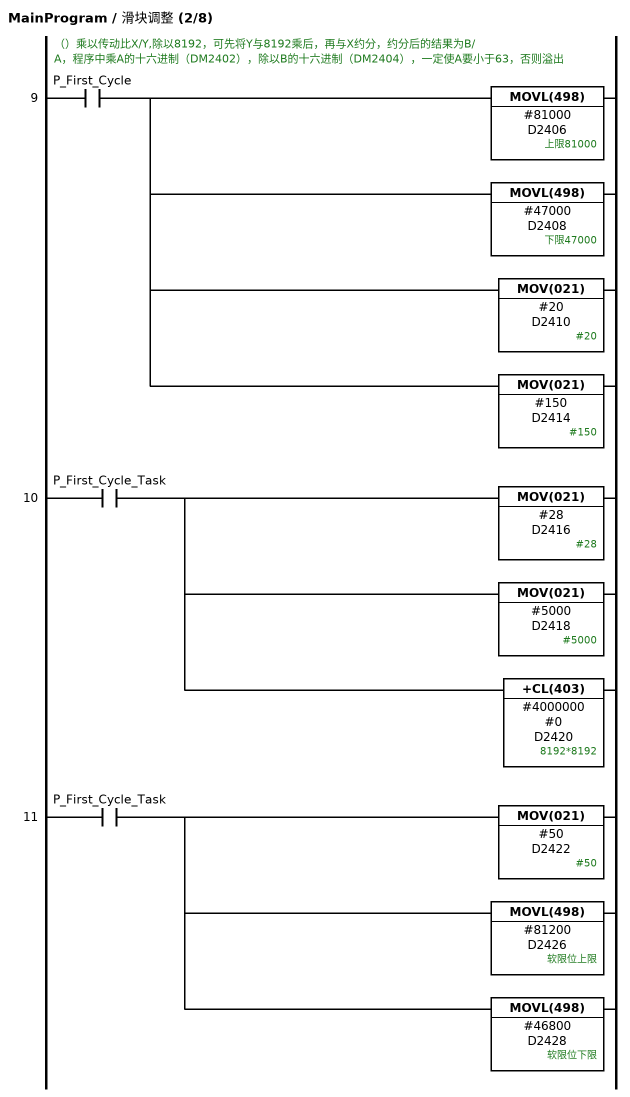
; [picture p24: MainProgram / 滑块调整, rungs 9-11]
; rung 9: （）乘以传动比X/Y,除以8192，可先将Y与8192乘后，再与X约分，约分后的结果为B/A，程序中乘A的十六进制（DM2402），除以B的十六进制（DM2404），一定使A要小于63，否则溢出
LD P_First_Cycle
MOVL(498) #81000 D2406  ; 上限81000
MOVL(498) #47000 D2408  ; 下限47000
MOV(021) #20 D2410  ; #20
MOV(021) #150 D2414  ; #150
; rung 10
LD P_First_Cycle_Task
MOV(021) #28 D2416  ; #28
MOV(021) #5000 D2418  ; #5000
+CL(403) #4000000 #0 D2420  ; 8192*8192
; rung 11
LD P_First_Cycle_Task
MOV(021) #50 D2422  ; #50
MOVL(498) #81200 D2426  ; 软限位上限
MOVL(498) #46800 D2428  ; 软限位下限

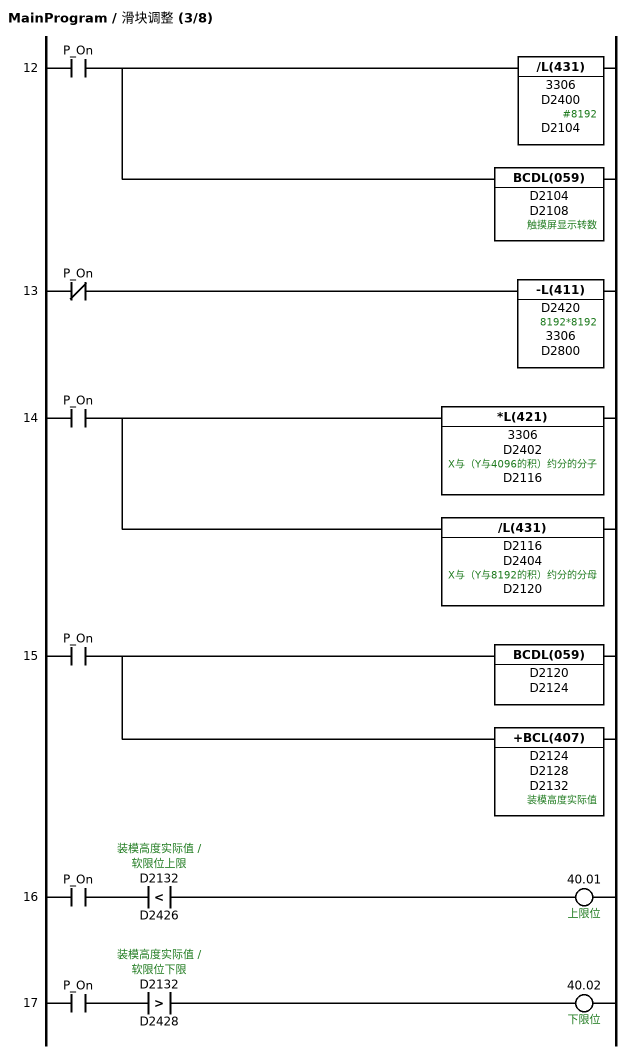
; rung 12
LD P_On
/L(431) 3306 D2400 D2104  ; #8192
BCDL(059) D2104 D2108  ; 触摸屏显示转数
; rung 13
LDNOT P_On
-L(411) D2420 3306 D2800  ; 8192*8192
; rung 14
LD P_On
*L(421) 3306 D2402 D2116  ; X与（Y与4096的积）约分的分子
/L(431) D2116 D2404 D2120  ; X与（Y与8192的积）约分的分母
; rung 15
LD P_On
BCDL(059) D2120 D2124
+BCL(407) D2124 D2128 D2132  ; 装模高度实际值
; rung 16
LD P_On
AND<L(311) D2132 D2426  ; 装模高度实际值, 软限位上限
OUT 40.01  ; 上限位
; rung 17
LD P_On
AND>L(321) D2132 D2428  ; 装模高度实际值, 软限位下限
OUT 40.02  ; 下限位

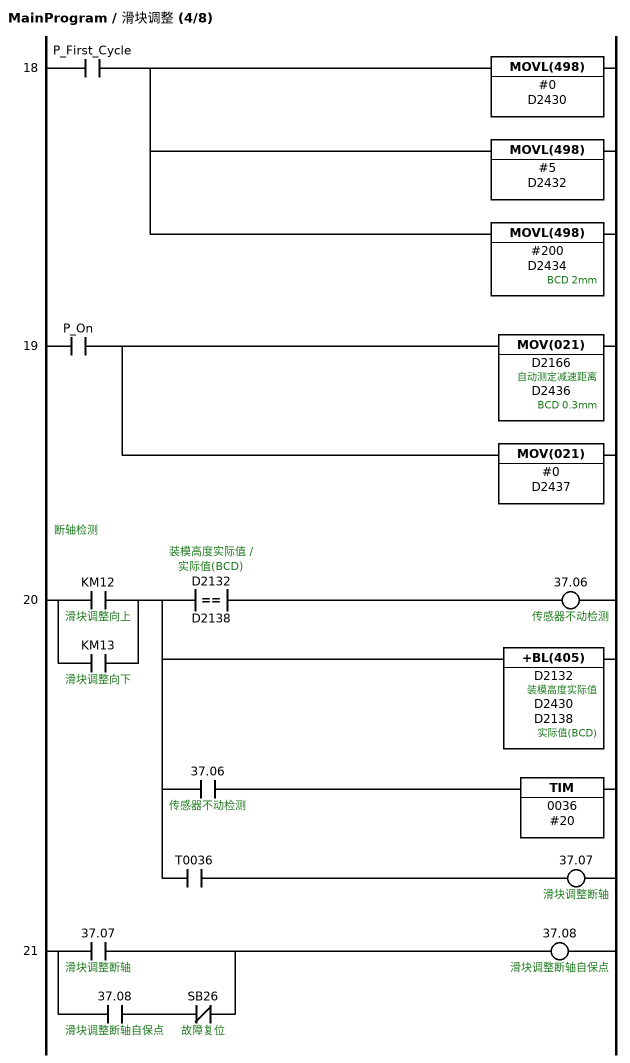
; rung 18
LD P_First_Cycle
MOVL(498) #0 D2430
MOVL(498) #5 D2432
MOVL(498) #200 D2434  ; BCD 2mm
; rung 19
LD P_On
MOV(021) D2166 D2436  ; 自动测定减速距离, BCD 0.3mm
MOV(021) #0 D2437
; rung 20: 断轴检测
LD KM12  ; 滑块调整向上
OR KM13  ; 滑块调整向下
OUT TR0
AND=L(301) D2132 D2138  ; 装模高度实际值, 实际值(BCD)
OUT 37.06  ; 传感器不动检测
LD TR0
+BL(405) D2132 D2430 D2138  ; 装模高度实际值, 实际值(BCD)
AND 37.06  ; 传感器不动检测
TIM 0036 #20
LD TR0
AND T0036
OUT 37.07  ; 滑块调整断轴
; rung 21
LD 37.07  ; 滑块调整断轴
LD 37.08  ; 滑块调整断轴自保点
ANDNOT SB26  ; 故障复位
ORLD
OUT 37.08  ; 滑块调整断轴自保点

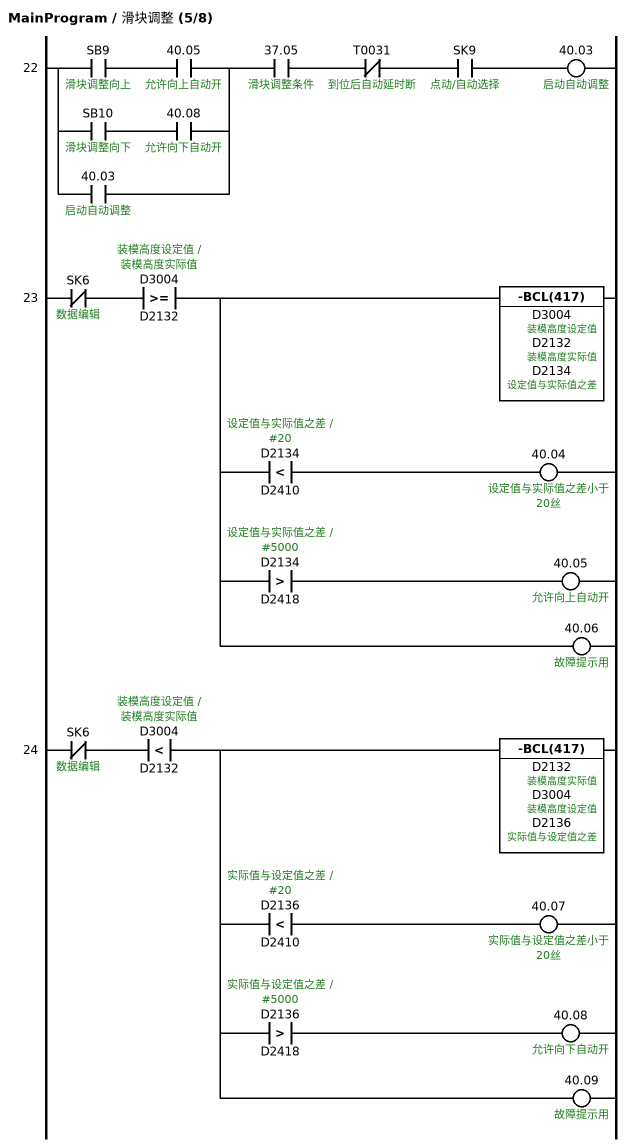
; rung 22
LD SB9  ; 滑块调整向上
AND 40.05  ; 允许向上自动开
LD SB10  ; 滑块调整向下
AND 40.08  ; 允许向下自动开
ORLD
OR 40.03  ; 启动自动调整
AND 37.05  ; 滑块调整条件
ANDNOT T0031  ; 到位后自动延时断
AND SK9  ; 点动/自动选择
OUT 40.03  ; 启动自动调整
; rung 23
LDNOT SK6  ; 数据编辑
AND>=L(326) D3004 D2132  ; 装模高度设定值, 装模高度实际值
OUT TR0
-BCL(417) D3004 D2132 D2134  ; 装模高度设定值, 装模高度实际值, 设定值与实际值之差
AND<L(311) D2134 D2410  ; 设定值与实际值之差, #20
OUT 40.04  ; 设定值与实际值之差小于20丝
LD TR0
AND>L(321) D2134 D2418  ; 设定值与实际值之差, #5000
OUT 40.05  ; 允许向上自动开
LD TR0
OUT 40.06  ; 故障提示用
; rung 24
LDNOT SK6  ; 数据编辑
AND<L(311) D3004 D2132  ; 装模高度设定值, 装模高度实际值
OUT TR0
-BCL(417) D2132 D3004 D2136  ; 装模高度实际值, 装模高度设定值, 实际值与设定值之差
AND<L(311) D2136 D2410  ; 实际值与设定值之差, #20
OUT 40.07  ; 实际值与设定值之差小于20丝
LD TR0
AND>L(321) D2136 D2418  ; 实际值与设定值之差, #5000
OUT 40.08  ; 允许向下自动开
LD TR0
OUT 40.09  ; 故障提示用

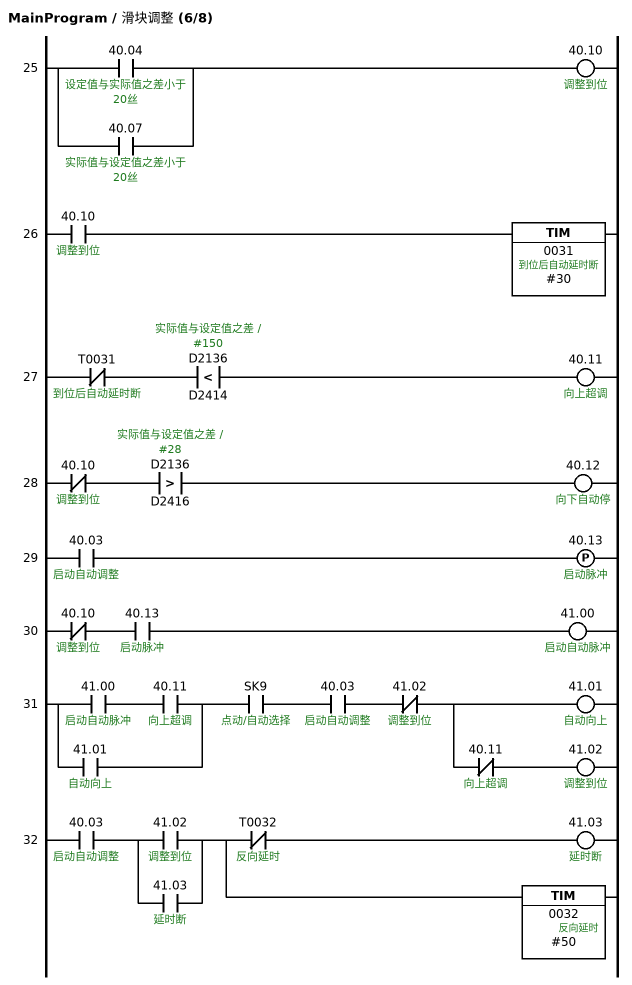
; rung 25
LD 40.04  ; 设定值与实际值之差小于20丝
OR 40.07  ; 实际值与设定值之差小于20丝
OUT 40.10  ; 调整到位
; rung 26
LD 40.10  ; 调整到位
TIM 0031 #30  ; 到位后自动延时断
; rung 27
LDNOT T0031  ; 到位后自动延时断
AND<L(311) D2136 D2414  ; 实际值与设定值之差, #150
OUT 40.11  ; 向上超调
; rung 28
LDNOT 40.10  ; 调整到位
AND>L(321) D2136 D2416  ; 实际值与设定值之差, #28
OUT 40.12  ; 向下自动停
; rung 29
LD 40.03  ; 启动自动调整
DIFU(013) 40.13  ; 启动脉冲
; rung 30
LDNOT 40.10  ; 调整到位
AND 40.13  ; 启动脉冲
OUT 41.00  ; 启动自动脉冲
; rung 31
LD 41.00  ; 启动自动脉冲
AND 40.11  ; 向上超调
OR 41.01  ; 自动向上
AND SK9  ; 点动/自动选择
AND 40.03  ; 启动自动调整
ANDNOT 41.02  ; 调整到位
OUT 41.01  ; 自动向上
ANDNOT 40.11  ; 向上超调
OUT 41.02  ; 调整到位
; rung 32
LD 40.03  ; 启动自动调整
LD 41.02  ; 调整到位
OR 41.03  ; 延时断
ANDLD
OUT TR0
ANDNOT T0032  ; 反向延时
OUT 41.03  ; 延时断
LD TR0
TIM 0032 #50  ; 反向延时

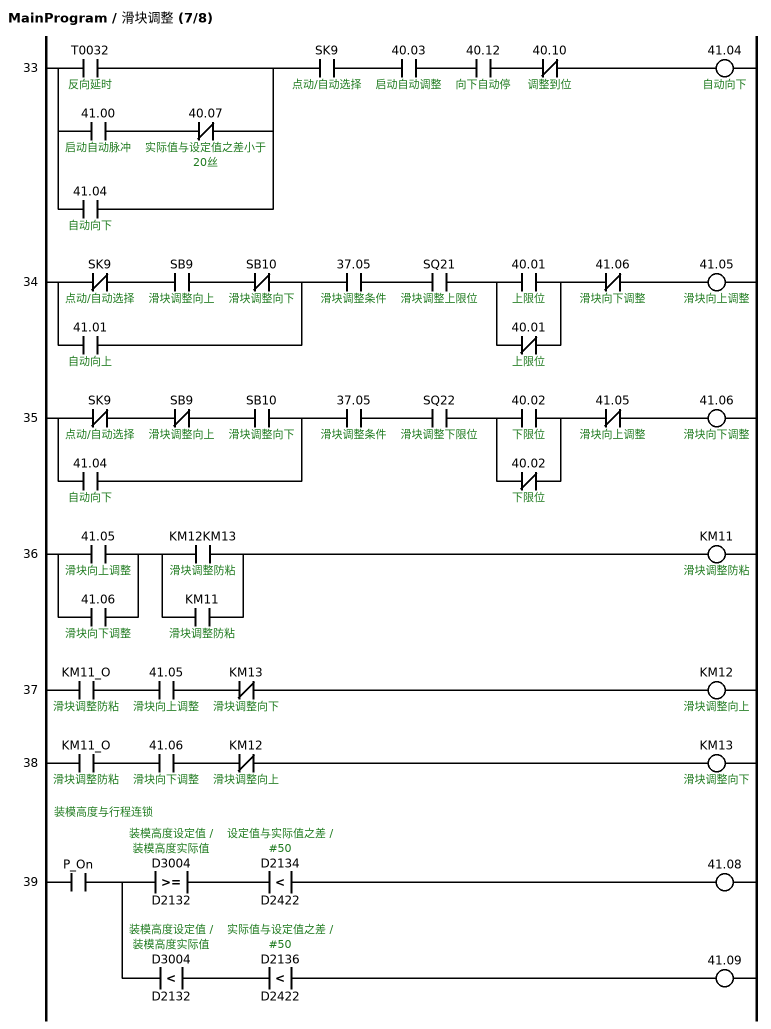
; rung 33
LD T0032  ; 反向延时
LD 41.00  ; 启动自动脉冲
ANDNOT 40.07  ; 实际值与设定值之差小于20丝
ORLD
OR 41.04  ; 自动向下
AND SK9  ; 点动/自动选择
AND 40.03  ; 启动自动调整
AND 40.12  ; 向下自动停
ANDNOT 40.10  ; 调整到位
OUT 41.04  ; 自动向下
; rung 34
LDNOT SK9  ; 点动/自动选择
AND SB9  ; 滑块调整向上
ANDNOT SB10  ; 滑块调整向下
OR 41.01  ; 自动向上
AND 37.05  ; 滑块调整条件
AND SQ21  ; 滑块调整上限位
LD 40.01  ; 上限位
ORNOT 40.01  ; 上限位
ANDLD
ANDNOT 41.06  ; 滑块向下调整
OUT 41.05  ; 滑块向上调整
; rung 35
LDNOT SK9  ; 点动/自动选择
ANDNOT SB9  ; 滑块调整向上
AND SB10  ; 滑块调整向下
OR 41.04  ; 自动向下
AND 37.05  ; 滑块调整条件
AND SQ22  ; 滑块调整下限位
LD 40.02  ; 下限位
ORNOT 40.02  ; 下限位
ANDLD
ANDNOT 41.05  ; 滑块向上调整
OUT 41.06  ; 滑块向下调整
; rung 36
LD 41.05  ; 滑块向上调整
OR 41.06  ; 滑块向下调整
LD KM12KM13  ; 滑块调整防粘
OR KM11  ; 滑块调整防粘
ANDLD
OUT KM11  ; 滑块调整防粘
; rung 37
LD KM11_O  ; 滑块调整防粘
AND 41.05  ; 滑块向上调整
ANDNOT KM13  ; 滑块调整向下
OUT KM12  ; 滑块调整向上
; rung 38
LD KM11_O  ; 滑块调整防粘
AND 41.06  ; 滑块向下调整
ANDNOT KM12  ; 滑块调整向上
OUT KM13  ; 滑块调整向下
; rung 39: 装模高度与行程连锁
LD P_On
OUT TR0
AND>=L(326) D3004 D2132  ; 装模高度设定值, 装模高度实际值
AND<L(311) D2134 D2422  ; 设定值与实际值之差, #50
OUT 41.08
LD TR0
AND<L(311) D3004 D2132  ; 装模高度设定值, 装模高度实际值
AND<L(311) D2136 D2422  ; 实际值与设定值之差, #50
OUT 41.09

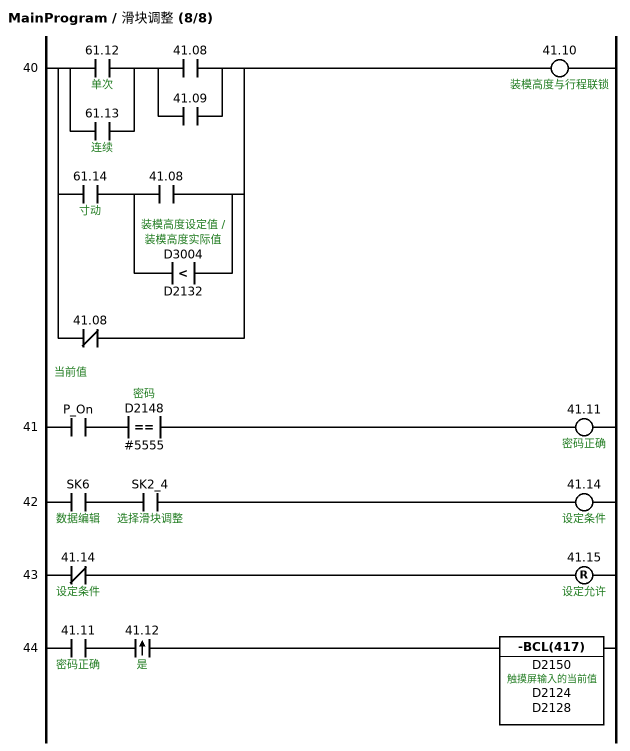
; rung 40
LD 61.12  ; 单次
OR 61.13  ; 连续
LD 41.08
OR 41.09
ANDLD
LD 61.14  ; 寸动
LD 41.08
OR<L(311) D3004 D2132  ; 装模高度设定值, 装模高度实际值
ANDLD
ORLD
ORNOT 41.08
OUT 41.10  ; 装模高度与行程联锁
; rung 41: 当前值
LD P_On
AND=(300) D2148 #5555  ; 密码
OUT 41.11  ; 密码正确
; rung 42
LD SK6  ; 数据编辑
AND SK2_4  ; 选择滑块调整
OUT 41.14  ; 设定条件
; rung 43
LDNOT 41.14  ; 设定条件
RSET 41.15  ; 设定允许
; rung 44
LD 41.11  ; 密码正确
@AND 41.12  ; 是
-BCL(417) D2150 D2124 D2128  ; 触摸屏输入的当前值

### Section 气垫调整

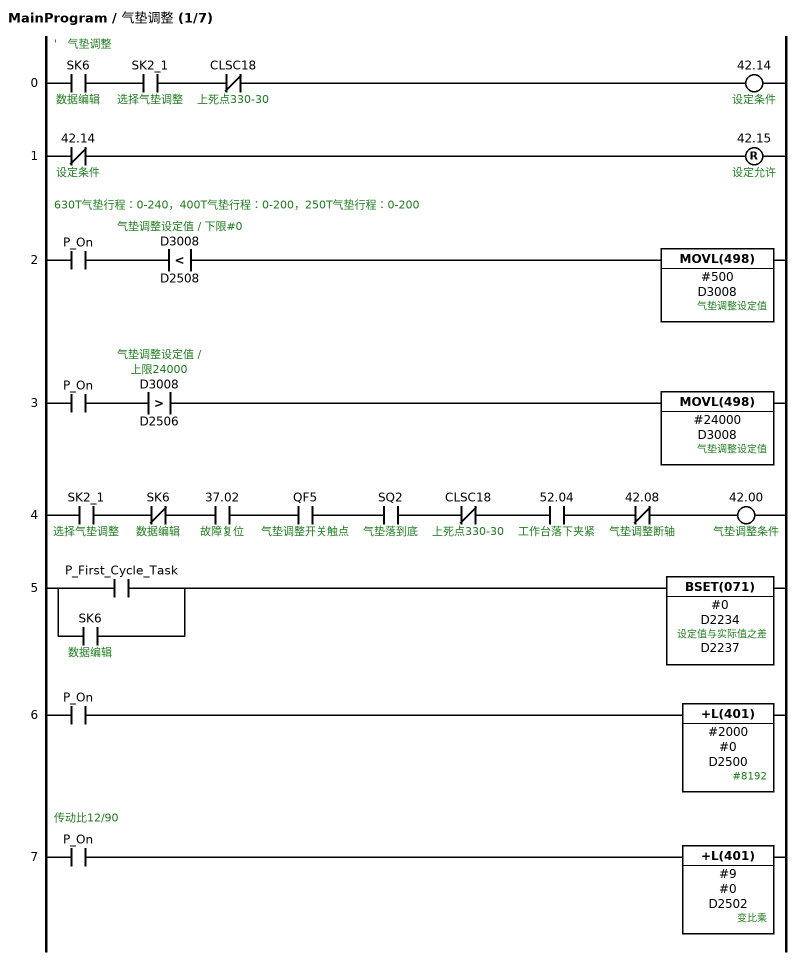
; rung 0: '   气垫调整
LD SK6  ; 数据编辑
AND SK2_1  ; 选择气垫调整
ANDNOT CLSC18  ; 上死点330-30
OUT 42.14  ; 设定条件
; rung 1
LDNOT 42.14  ; 设定条件
RSET 42.15  ; 设定允许
; rung 2: 630T气垫行程：0-240，400T气垫行程：0-200，250T气垫行程：0-200
LD P_On
AND<L(311) D3008 D2508  ; 气垫调整设定值, 下限#0
MOVL(498) #500 D3008  ; 气垫调整设定值
; rung 3
LD P_On
AND>L(321) D3008 D2506  ; 气垫调整设定值, 上限24000
MOVL(498) #24000 D3008  ; 气垫调整设定值
; rung 4
LD SK2_1  ; 选择气垫调整
ANDNOT SK6  ; 数据编辑
AND 37.02  ; 故障复位
AND QF5  ; 气垫调整开关触点
AND SQ2  ; 气垫落到底
ANDNOT CLSC18  ; 上死点330-30
AND 52.04  ; 工作台落下夹紧
ANDNOT 42.08  ; 气垫调整断轴
OUT 42.00  ; 气垫调整条件
; rung 5
LD P_First_Cycle_Task
OR SK6  ; 数据编辑
BSET(071) #0 D2234 D2237  ; 设定值与实际值之差
; rung 6
LD P_On
+L(401) #2000 #0 D2500  ; #8192
; rung 7: 传动比12/90
LD P_On
+L(401) #9 #0 D2502  ; 变比乘

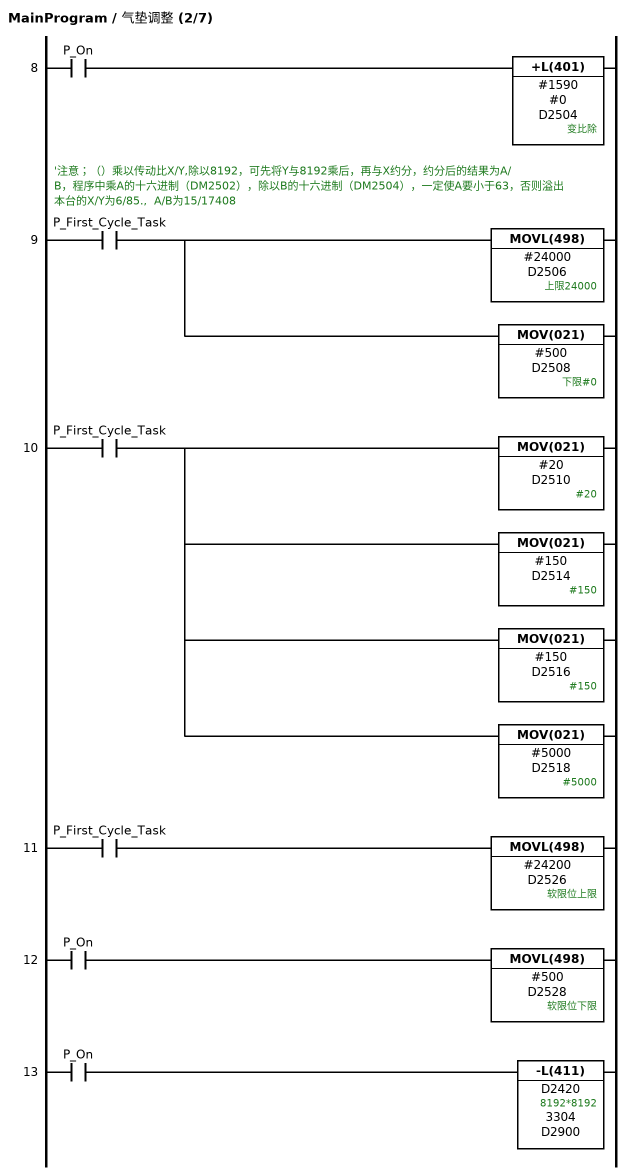
; rung 8
LD P_On
+L(401) #1590 #0 D2504  ; 变比除
; rung 9: '注意；（）乘以传动比X/Y,除以8192，可先将Y与8192乘后，再与X约分，约分后的结果为A/B，程序中乘A的十六进制（DM2502），除以B的十六进制（DM2504），一定使A要小于63，否则溢出                本台的X/Y为6/85.,  A/B为15/17408
LD P_First_Cycle_Task
MOVL(498) #24000 D2506  ; 上限24000
MOV(021) #500 D2508  ; 下限#0
; rung 10
LD P_First_Cycle_Task
MOV(021) #20 D2510  ; #20
MOV(021) #150 D2514  ; #150
MOV(021) #150 D2516  ; #150
MOV(021) #5000 D2518  ; #5000
; rung 11
LD P_First_Cycle_Task
MOVL(498) #24200 D2526  ; 软限位上限
; rung 12
LD P_On
MOVL(498) #500 D2528  ; 软限位下限
; rung 13
LD P_On
-L(411) D2420 3304 D2900  ; 8192*8192

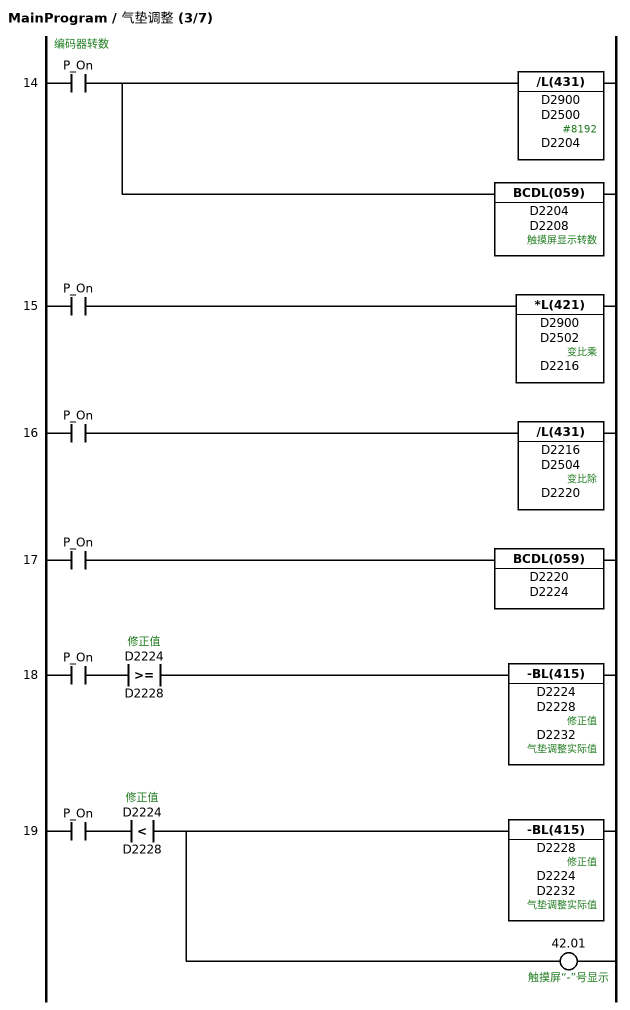
; rung 14: 编码器转数
LD P_On
/L(431) D2900 D2500 D2204  ; #8192
BCDL(059) D2204 D2208  ; 触摸屏显示转数
; rung 15
LD P_On
*L(421) D2900 D2502 D2216  ; 变比乘
; rung 16
LD P_On
/L(431) D2216 D2504 D2220  ; 变比除
; rung 17
LD P_On
BCDL(059) D2220 D2224
; rung 18
LD P_On
AND>=L(326) D2224 D2228  ; 修正值
-BL(415) D2224 D2228 D2232  ; 修正值, 气垫调整实际值
; rung 19
LD P_On
AND<L(311) D2224 D2228  ; 修正值
-BL(415) D2228 D2224 D2232  ; 修正值, 气垫调整实际值
OUT 42.01  ; 触摸屏“-”号显示

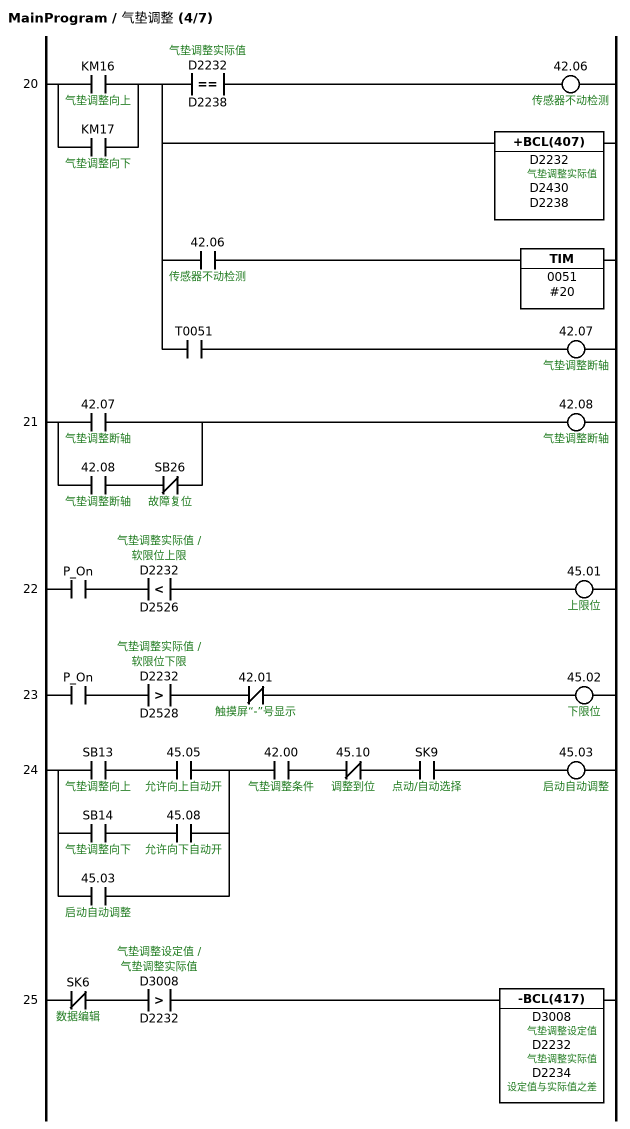
; rung 20
LD KM16  ; 气垫调整向上
OR KM17  ; 气垫调整向下
OUT TR0
AND=L(301) D2232 D2238  ; 气垫调整实际值
OUT 42.06  ; 传感器不动检测
LD TR0
+BCL(407) D2232 D2430 D2238  ; 气垫调整实际值
AND 42.06  ; 传感器不动检测
TIM 0051 #20
LD TR0
AND T0051
OUT 42.07  ; 气垫调整断轴
; rung 21
LD 42.07  ; 气垫调整断轴
LD 42.08  ; 气垫调整断轴
ANDNOT SB26  ; 故障复位
ORLD
OUT 42.08  ; 气垫调整断轴
; rung 22
LD P_On
AND<L(311) D2232 D2526  ; 气垫调整实际值, 软限位上限
OUT 45.01  ; 上限位
; rung 23
LD P_On
AND>L(321) D2232 D2528  ; 气垫调整实际值, 软限位下限
ANDNOT 42.01  ; 触摸屏“-”号显示
OUT 45.02  ; 下限位
; rung 24
LD SB13  ; 气垫调整向上
AND 45.05  ; 允许向上自动开
LD SB14  ; 气垫调整向下
AND 45.08  ; 允许向下自动开
ORLD
OR 45.03  ; 启动自动调整
AND 42.00  ; 气垫调整条件
ANDNOT 45.10  ; 调整到位
AND SK9  ; 点动/自动选择
OUT 45.03  ; 启动自动调整
; rung 25
LDNOT SK6  ; 数据编辑
AND>L(321) D3008 D2232  ; 气垫调整设定值, 气垫调整实际值
-BCL(417) D3008 D2232 D2234  ; 气垫调整设定值, 气垫调整实际值, 设定值与实际值之差

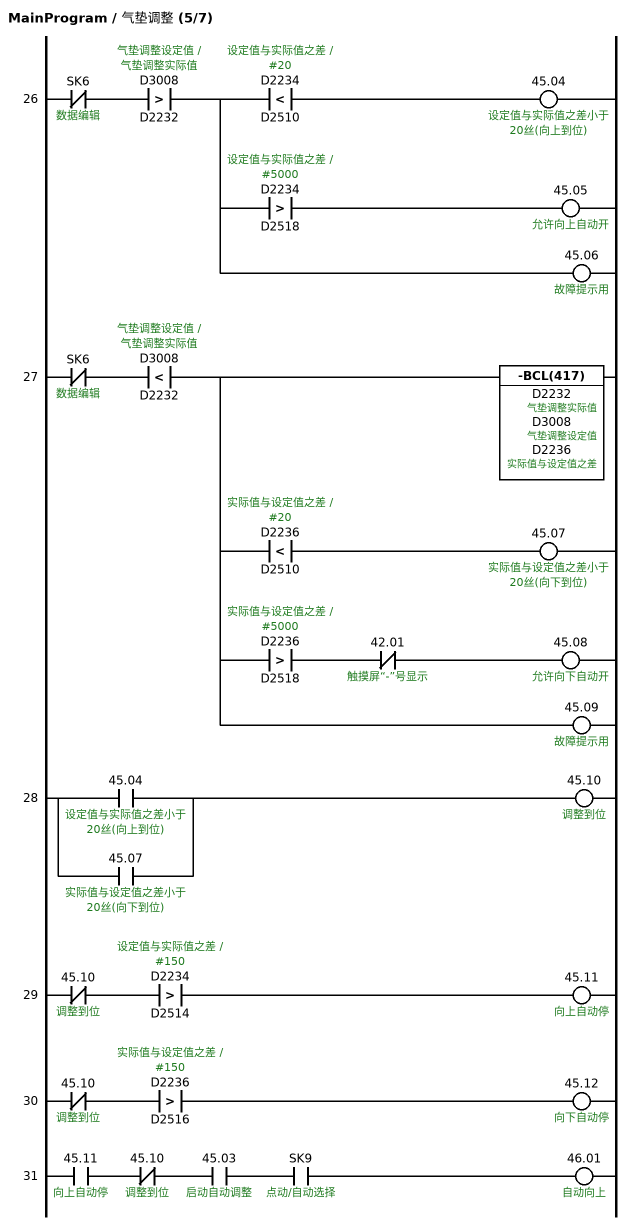
; rung 26
LDNOT SK6  ; 数据编辑
AND>L(321) D3008 D2232  ; 气垫调整设定值, 气垫调整实际值
OUT TR0
AND<L(311) D2234 D2510  ; 设定值与实际值之差, #20
OUT 45.04  ; 设定值与实际值之差小于20丝(向上到位)
LD TR0
AND>L(321) D2234 D2518  ; 设定值与实际值之差, #5000
OUT 45.05  ; 允许向上自动开
LD TR0
OUT 45.06  ; 故障提示用
; rung 27
LDNOT SK6  ; 数据编辑
AND<L(311) D3008 D2232  ; 气垫调整设定值, 气垫调整实际值
OUT TR0
-BCL(417) D2232 D3008 D2236  ; 气垫调整实际值, 气垫调整设定值, 实际值与设定值之差
AND<L(311) D2236 D2510  ; 实际值与设定值之差, #20
OUT 45.07  ; 实际值与设定值之差小于20丝(向下到位)
LD TR0
AND>L(321) D2236 D2518  ; 实际值与设定值之差, #5000
ANDNOT 42.01  ; 触摸屏“-”号显示
OUT 45.08  ; 允许向下自动开
LD TR0
OUT 45.09  ; 故障提示用
; rung 28
LD 45.04  ; 设定值与实际值之差小于20丝(向上到位)
OR 45.07  ; 实际值与设定值之差小于20丝(向下到位)
OUT 45.10  ; 调整到位
; rung 29
LDNOT 45.10  ; 调整到位
AND>L(321) D2234 D2514  ; 设定值与实际值之差, #150
OUT 45.11  ; 向上自动停
; rung 30
LDNOT 45.10  ; 调整到位
AND>L(321) D2236 D2516  ; 实际值与设定值之差, #150
OUT 45.12  ; 向下自动停
; rung 31
LD 45.11  ; 向上自动停
ANDNOT 45.10  ; 调整到位
AND 45.03  ; 启动自动调整
AND SK9  ; 点动/自动选择
OUT 46.01  ; 自动向上

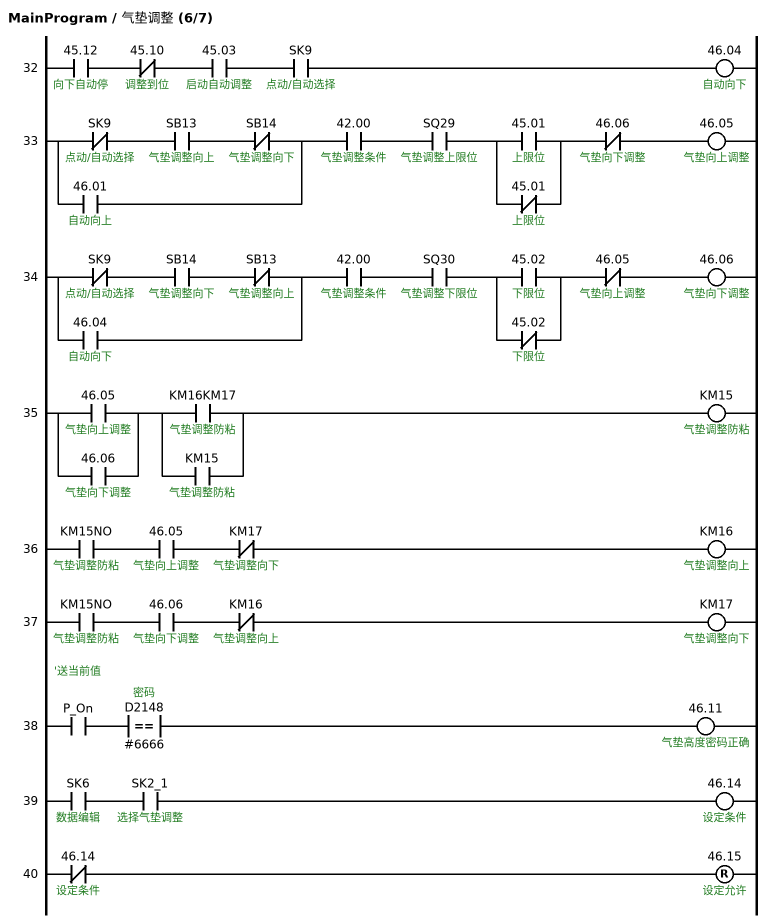
; rung 32
LD 45.12  ; 向下自动停
ANDNOT 45.10  ; 调整到位
AND 45.03  ; 启动自动调整
AND SK9  ; 点动/自动选择
OUT 46.04  ; 自动向下
; rung 33
LDNOT SK9  ; 点动/自动选择
AND SB13  ; 气垫调整向上
ANDNOT SB14  ; 气垫调整向下
OR 46.01  ; 自动向上
AND 42.00  ; 气垫调整条件
AND SQ29  ; 气垫调整上限位
LD 45.01  ; 上限位
ORNOT 45.01  ; 上限位
ANDLD
ANDNOT 46.06  ; 气垫向下调整
OUT 46.05  ; 气垫向上调整
; rung 34
LDNOT SK9  ; 点动/自动选择
AND SB14  ; 气垫调整向下
ANDNOT SB13  ; 气垫调整向上
OR 46.04  ; 自动向下
AND 42.00  ; 气垫调整条件
AND SQ30  ; 气垫调整下限位
LD 45.02  ; 下限位
ORNOT 45.02  ; 下限位
ANDLD
ANDNOT 46.05  ; 气垫向上调整
OUT 46.06  ; 气垫向下调整
; rung 35
LD 46.05  ; 气垫向上调整
OR 46.06  ; 气垫向下调整
LD KM16KM17  ; 气垫调整防粘
OR KM15  ; 气垫调整防粘
ANDLD
OUT KM15  ; 气垫调整防粘
; rung 36
LD KM15NO  ; 气垫调整防粘
AND 46.05  ; 气垫向上调整
ANDNOT KM17  ; 气垫调整向下
OUT KM16  ; 气垫调整向上
; rung 37
LD KM15NO  ; 气垫调整防粘
AND 46.06  ; 气垫向下调整
ANDNOT KM16  ; 气垫调整向上
OUT KM17  ; 气垫调整向下
; rung 38: '送当前值
LD P_On
AND=L(301) D2148 #6666  ; 密码
OUT 46.11  ; 气垫高度密码正确
; rung 39
LD SK6  ; 数据编辑
AND SK2_1  ; 选择气垫调整
OUT 46.14  ; 设定条件
; rung 40
LDNOT 46.14  ; 设定条件
RSET 46.15  ; 设定允许

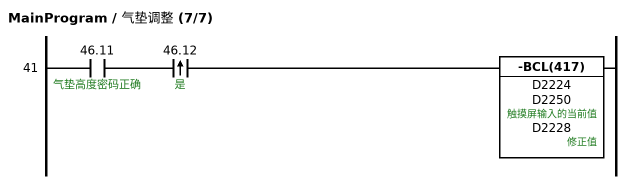
; rung 41
LD 46.11  ; 气垫高度密码正确
@AND 46.12  ; 是
-BCL(417) D2224 D2250 D2228  ; 触摸屏输入的当前值, 修正值

### Section 气垫顶起

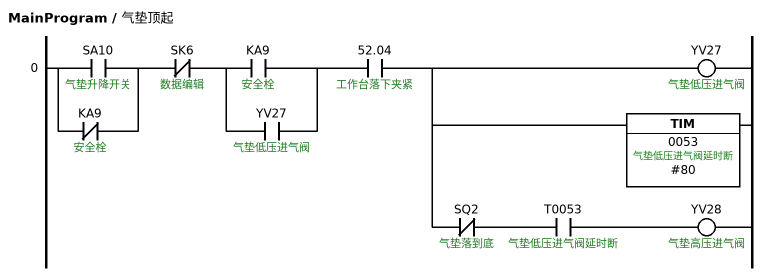
; rung 0
LD SA10  ; 气垫升降开关
ORNOT KA9  ; 安全栓
ANDNOT SK6  ; 数据编辑
LD KA9  ; 安全栓
OR YV27  ; 气垫低压进气阀
ANDLD
AND 52.04  ; 工作台落下夹紧
OUT YV27  ; 气垫低压进气阀
TIM 0053 #80  ; 气垫低压进气阀延时断
ANDNOT SQ2  ; 气垫落到底
AND T0053  ; 气垫低压进气阀延时断
OUT YV28  ; 气垫高压进气阀

### Section 工作台

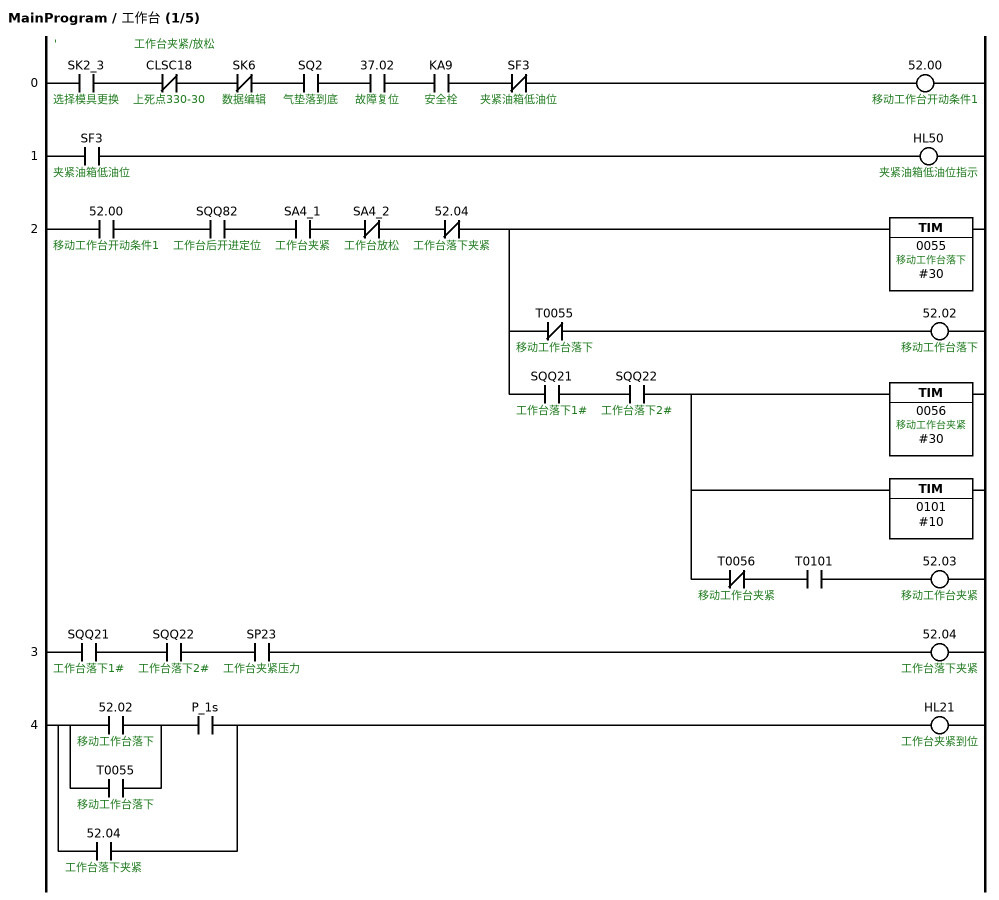
; rung 0: '                      工作台夹紧/放松
LD SK2_3  ; 选择模具更换
ANDNOT CLSC18  ; 上死点330-30
ANDNOT SK6  ; 数据编辑
AND SQ2  ; 气垫落到底
AND 37.02  ; 故障复位
AND KA9  ; 安全栓
ANDNOT SF3  ; 夹紧油箱低油位
OUT 52.00  ; 移动工作台开动条件1
; rung 1
LD SF3  ; 夹紧油箱低油位
OUT HL50  ; 夹紧油箱低油位指示
; rung 2
LD 52.00  ; 移动工作台开动条件1
AND SQQ82  ; 工作台后开进定位
AND SA4_1  ; 工作台夹紧
ANDNOT SA4_2  ; 工作台放松
ANDNOT 52.04  ; 工作台落下夹紧
OUT TR0
TIM 0055 #30  ; 移动工作台落下
ANDNOT T0055  ; 移动工作台落下
OUT 52.02  ; 移动工作台落下
LD TR0
AND SQQ21  ; 工作台落下1#
AND SQQ22  ; 工作台落下2#
TIM 0056 #30  ; 移动工作台夹紧
TIM 0101 #10
ANDNOT T0056  ; 移动工作台夹紧
AND T0101
OUT 52.03  ; 移动工作台夹紧
; rung 3
LD SQQ21  ; 工作台落下1#
AND SQQ22  ; 工作台落下2#
AND SP23  ; 工作台夹紧压力
OUT 52.04  ; 工作台落下夹紧
; rung 4
LD 52.02  ; 移动工作台落下
OR T0055  ; 移动工作台落下
AND P_1s
OR 52.04  ; 工作台落下夹紧
OUT HL21  ; 工作台夹紧到位

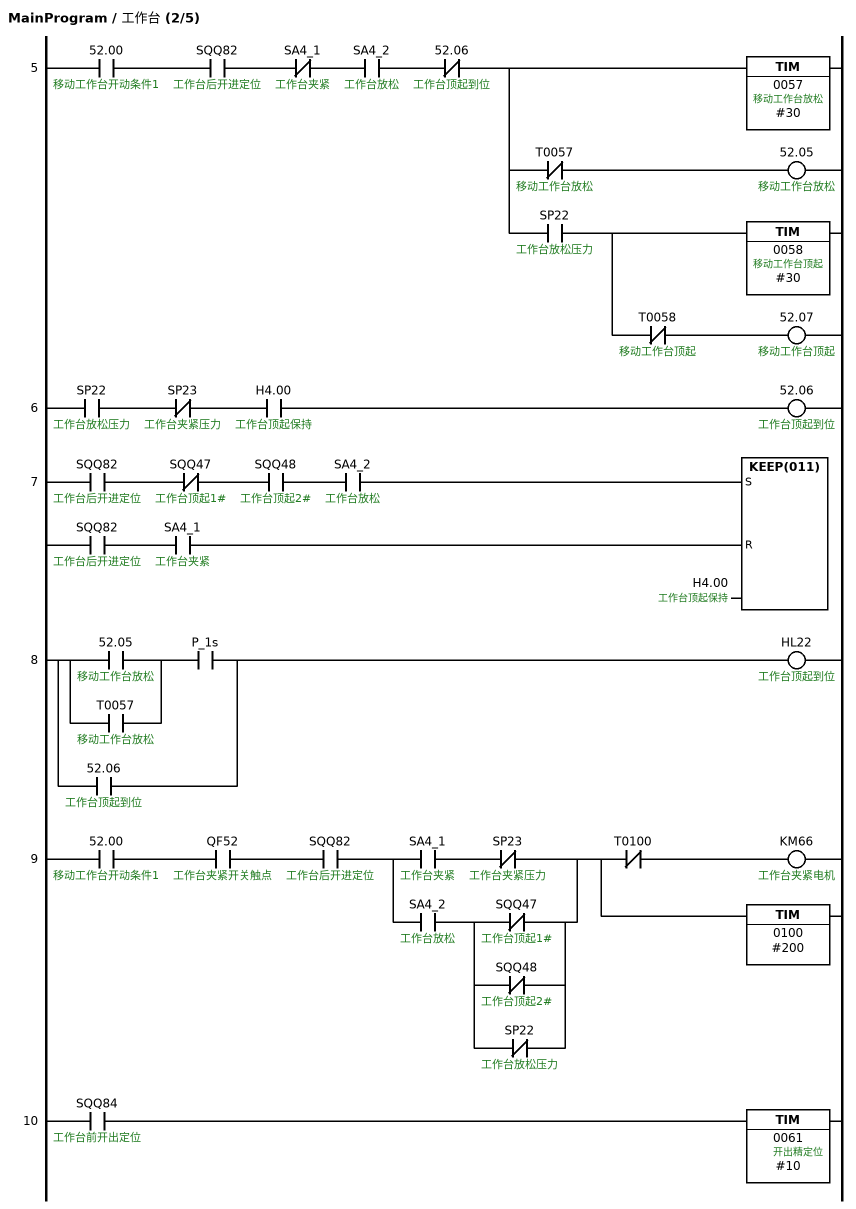
; rung 5
LD 52.00  ; 移动工作台开动条件1
AND SQQ82  ; 工作台后开进定位
ANDNOT SA4_1  ; 工作台夹紧
AND SA4_2  ; 工作台放松
ANDNOT 52.06  ; 工作台顶起到位
OUT TR0
TIM 0057 #30  ; 移动工作台放松
ANDNOT T0057  ; 移动工作台放松
OUT 52.05  ; 移动工作台放松
LD TR0
AND SP22  ; 工作台放松压力
TIM 0058 #30  ; 移动工作台顶起
ANDNOT T0058  ; 移动工作台顶起
OUT 52.07  ; 移动工作台顶起
; rung 6
LD SP22  ; 工作台放松压力
ANDNOT SP23  ; 工作台夹紧压力
AND H4.00  ; 工作台顶起保持
OUT 52.06  ; 工作台顶起到位
; rung 7
LD SQQ82  ; 工作台后开进定位
ANDNOT SQQ47  ; 工作台顶起1#
AND SQQ48  ; 工作台顶起2#
AND SA4_2  ; 工作台放松
LD SQQ82  ; 工作台后开进定位
AND SA4_1  ; 工作台夹紧
KEEP(011) H4.00  ; 工作台顶起保持
; rung 8
LD 52.05  ; 移动工作台放松
OR T0057  ; 移动工作台放松
AND P_1s
OR 52.06  ; 工作台顶起到位
OUT HL22  ; 工作台顶起到位
; rung 9
LD 52.00  ; 移动工作台开动条件1
AND QF52  ; 工作台夹紧开关触点
AND SQQ82  ; 工作台后开进定位
LD SA4_1  ; 工作台夹紧
ANDNOT SP23  ; 工作台夹紧压力
LD SA4_2  ; 工作台放松
LDNOT SQQ47  ; 工作台顶起1#
ORNOT SQQ48  ; 工作台顶起2#
ORNOT SP22  ; 工作台放松压力
ANDLD
ORLD
ANDLD
OUT TR0
ANDNOT T0100
OUT KM66  ; 工作台夹紧电机
LD TR0
TIM 0100 #200
; rung 10
LD SQQ84  ; 工作台前开出定位
TIM 0061 #10  ; 开出精定位

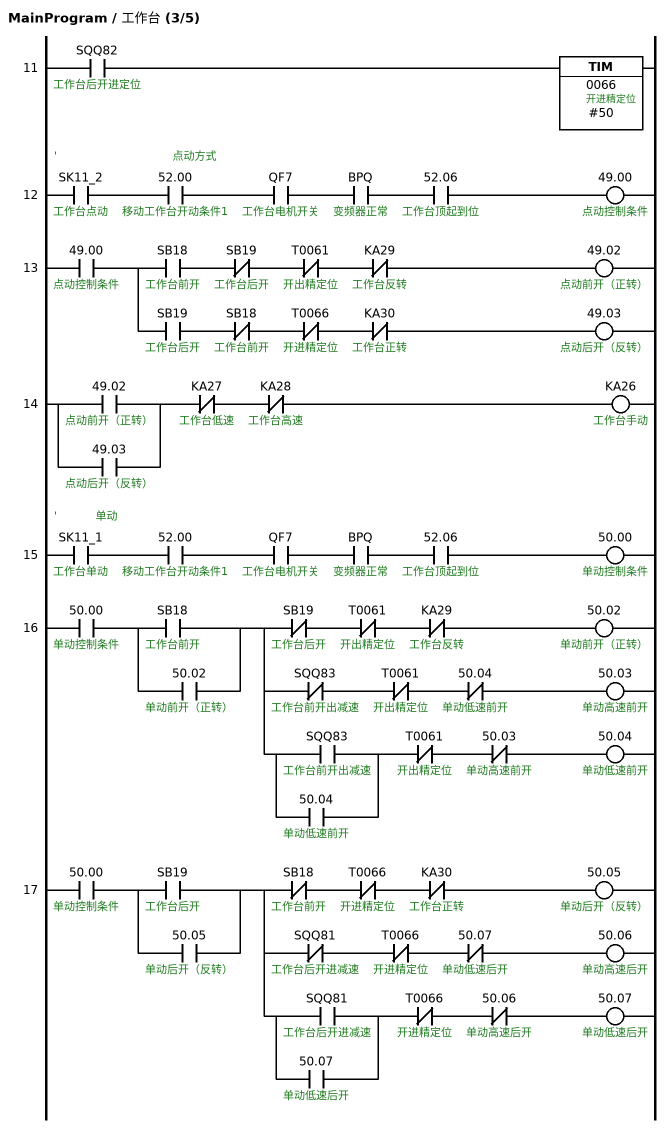
; rung 11
LD SQQ82  ; 工作台后开进定位
TIM 0066 #50  ; 开进精定位
; rung 12: '                                 点动方式
LD SK11_2  ; 工作台点动
AND 52.00  ; 移动工作台开动条件1
AND QF7  ; 工作台电机开关
AND BPQ  ; 变频器正常
AND 52.06  ; 工作台顶起到位
OUT 49.00  ; 点动控制条件
; rung 13
LD 49.00  ; 点动控制条件
OUT TR0
AND SB18  ; 工作台前开
ANDNOT SB19  ; 工作台后开
ANDNOT T0061  ; 开出精定位
ANDNOT KA29  ; 工作台反转
OUT 49.02  ; 点动前开（正转）
LD TR0
AND SB19  ; 工作台后开
ANDNOT SB18  ; 工作台前开
ANDNOT T0066  ; 开进精定位
ANDNOT KA30  ; 工作台正转
OUT 49.03  ; 点动后开（反转）
; rung 14
LD 49.02  ; 点动前开（正转）
OR 49.03  ; 点动后开（反转）
ANDNOT KA27  ; 工作台低速
ANDNOT KA28  ; 工作台高速
OUT KA26  ; 工作台手动
; rung 15: '           单动
LD SK11_1  ; 工作台单动
AND 52.00  ; 移动工作台开动条件1
AND QF7  ; 工作台电机开关
AND BPQ  ; 变频器正常
AND 52.06  ; 工作台顶起到位
OUT 50.00  ; 单动控制条件
; rung 16
LD 50.00  ; 单动控制条件
LD SB18  ; 工作台前开
OR 50.02  ; 单动前开（正转）
ANDLD
OUT TR0
ANDNOT SB19  ; 工作台后开
ANDNOT T0061  ; 开出精定位
ANDNOT KA29  ; 工作台反转
OUT 50.02  ; 单动前开（正转）
LD TR0
ANDNOT SQQ83  ; 工作台前开出减速
ANDNOT T0061  ; 开出精定位
ANDNOT 50.04  ; 单动低速前开
OUT 50.03  ; 单动高速前开
LD TR0
LD SQQ83  ; 工作台前开出减速
OR 50.04  ; 单动低速前开
ANDLD
ANDNOT T0061  ; 开出精定位
ANDNOT 50.03  ; 单动高速前开
OUT 50.04  ; 单动低速前开
; rung 17
LD 50.00  ; 单动控制条件
LD SB19  ; 工作台后开
OR 50.05  ; 单动后开（反转）
ANDLD
OUT TR0
ANDNOT SB18  ; 工作台前开
ANDNOT T0066  ; 开进精定位
ANDNOT KA30  ; 工作台正转
OUT 50.05  ; 单动后开（反转）
LD TR0
ANDNOT SQQ81  ; 工作台后开进减速
ANDNOT T0066  ; 开进精定位
ANDNOT 50.07  ; 单动低速后开
OUT 50.06  ; 单动高速后开
LD TR0
LD SQQ81  ; 工作台后开进减速
OR 50.07  ; 单动低速后开
ANDLD
ANDNOT T0066  ; 开进精定位
ANDNOT 50.06  ; 单动高速后开
OUT 50.07  ; 单动低速后开

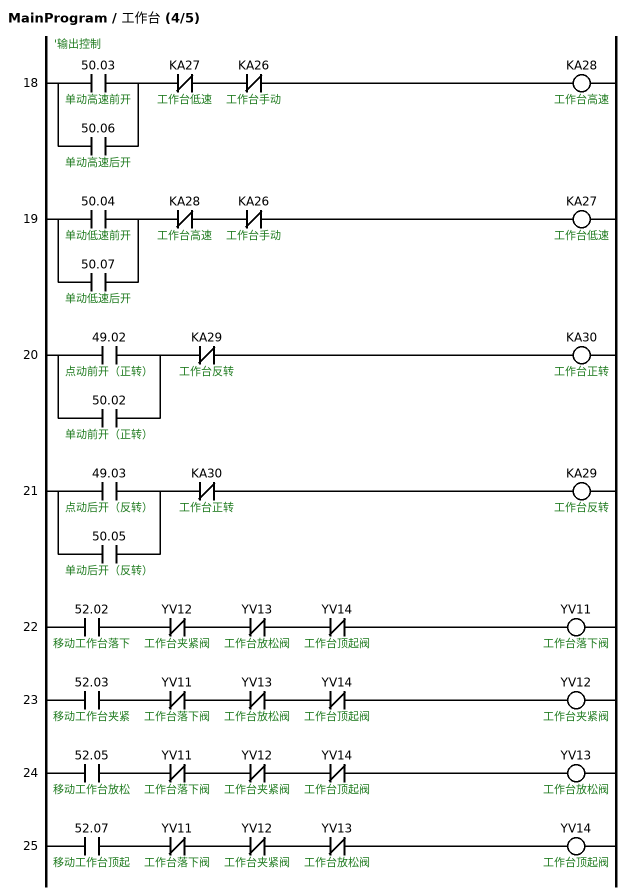
; rung 18: '输出控制
LD 50.03  ; 单动高速前开
OR 50.06  ; 单动高速后开
ANDNOT KA27  ; 工作台低速
ANDNOT KA26  ; 工作台手动
OUT KA28  ; 工作台高速
; rung 19
LD 50.04  ; 单动低速前开
OR 50.07  ; 单动低速后开
ANDNOT KA28  ; 工作台高速
ANDNOT KA26  ; 工作台手动
OUT KA27  ; 工作台低速
; rung 20
LD 49.02  ; 点动前开（正转）
OR 50.02  ; 单动前开（正转）
ANDNOT KA29  ; 工作台反转
OUT KA30  ; 工作台正转
; rung 21
LD 49.03  ; 点动后开（反转）
OR 50.05  ; 单动后开（反转）
ANDNOT KA30  ; 工作台正转
OUT KA29  ; 工作台反转
; rung 22
LD 52.02  ; 移动工作台落下
ANDNOT YV12  ; 工作台夹紧阀
ANDNOT YV13  ; 工作台放松阀
ANDNOT YV14  ; 工作台顶起阀
OUT YV11  ; 工作台落下阀
; rung 23
LD 52.03  ; 移动工作台夹紧
ANDNOT YV11  ; 工作台落下阀
ANDNOT YV13  ; 工作台放松阀
ANDNOT YV14  ; 工作台顶起阀
OUT YV12  ; 工作台夹紧阀
; rung 24
LD 52.05  ; 移动工作台放松
ANDNOT YV11  ; 工作台落下阀
ANDNOT YV12  ; 工作台夹紧阀
ANDNOT YV14  ; 工作台顶起阀
OUT YV13  ; 工作台放松阀
; rung 25
LD 52.07  ; 移动工作台顶起
ANDNOT YV11  ; 工作台落下阀
ANDNOT YV12  ; 工作台夹紧阀
ANDNOT YV13  ; 工作台放松阀
OUT YV14  ; 工作台顶起阀

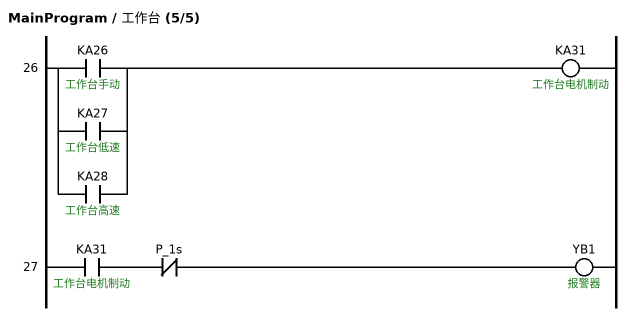
; rung 26
LD KA26  ; 工作台手动
OR KA27  ; 工作台低速
OR KA28  ; 工作台高速
OUT KA31  ; 工作台电机制动
; rung 27
LD KA31  ; 工作台电机制动
ANDNOT P_1s
OUT YB1  ; 报警器

### Section 自动化气源

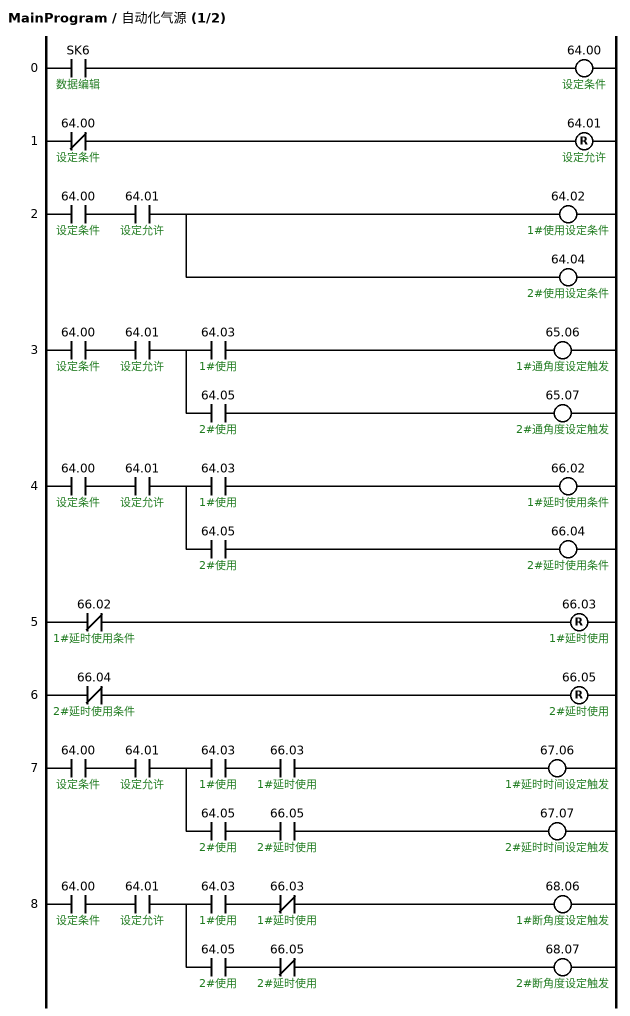
; rung 0
LD SK6  ; 数据编辑
OUT 64.00  ; 设定条件
; rung 1
LDNOT 64.00  ; 设定条件
RSET 64.01  ; 设定允许
; rung 2
LD 64.00  ; 设定条件
AND 64.01  ; 设定允许
OUT 64.02  ; 1#使用设定条件
OUT 64.04  ; 2#使用设定条件
; rung 3
LD 64.00  ; 设定条件
AND 64.01  ; 设定允许
OUT TR0
AND 64.03  ; 1#使用
OUT 65.06  ; 1#通角度设定触发
LD TR0
AND 64.05  ; 2#使用
OUT 65.07  ; 2#通角度设定触发
; rung 4
LD 64.00  ; 设定条件
AND 64.01  ; 设定允许
OUT TR0
AND 64.03  ; 1#使用
OUT 66.02  ; 1#延时使用条件
LD TR0
AND 64.05  ; 2#使用
OUT 66.04  ; 2#延时使用条件
; rung 5
LDNOT 66.02  ; 1#延时使用条件
RSET 66.03  ; 1#延时使用
; rung 6
LDNOT 66.04  ; 2#延时使用条件
RSET 66.05  ; 2#延时使用
; rung 7
LD 64.00  ; 设定条件
AND 64.01  ; 设定允许
OUT TR0
AND 64.03  ; 1#使用
AND 66.03  ; 1#延时使用
OUT 67.06  ; 1#延时时间设定触发
LD TR0
AND 64.05  ; 2#使用
AND 66.05  ; 2#延时使用
OUT 67.07  ; 2#延时时间设定触发
; rung 8
LD 64.00  ; 设定条件
AND 64.01  ; 设定允许
OUT TR0
AND 64.03  ; 1#使用
ANDNOT 66.03  ; 1#延时使用
OUT 68.06  ; 1#断角度设定触发
LD TR0
AND 64.05  ; 2#使用
ANDNOT 66.05  ; 2#延时使用
OUT 68.07  ; 2#断角度设定触发

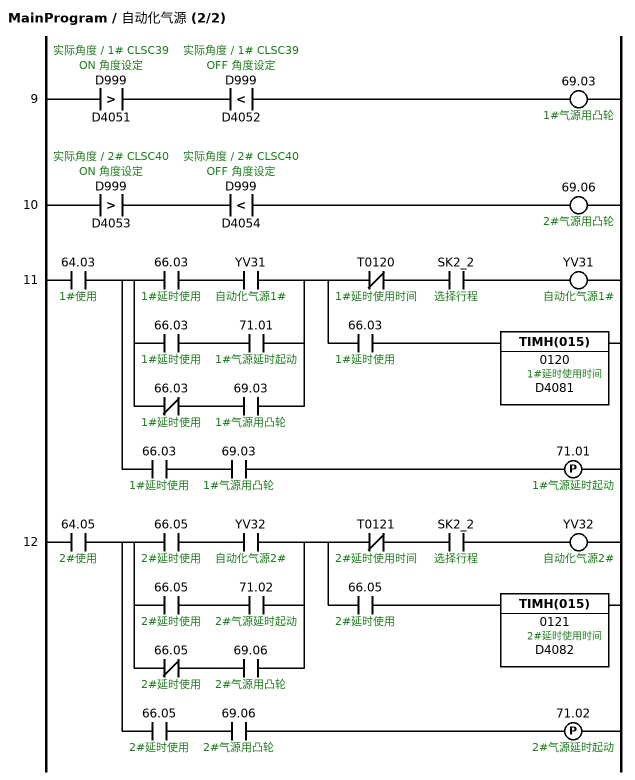
; rung 9
LD>(320) D999 D4051  ; 实际角度, 1# CLSC39 ON 角度设定
AND<(310) D999 D4052  ; 实际角度, 1# CLSC39 OFF 角度设定
OUT 69.03  ; 1#气源用凸轮
; rung 10
LD>(320) D999 D4053  ; 实际角度, 2# CLSC40 ON 角度设定
AND<(310) D999 D4054  ; 实际角度, 2# CLSC40 OFF 角度设定
OUT 69.06  ; 2#气源用凸轮
; rung 11
LD 64.03  ; 1#使用
OUT TR0
LD 66.03  ; 1#延时使用
AND YV31  ; 自动化气源1#
LD 66.03  ; 1#延时使用
AND 71.01  ; 1#气源延时起动
ORLD
LDNOT 66.03  ; 1#延时使用
AND 69.03  ; 1#气源用凸轮
ORLD
ANDLD
OUT TR1
ANDNOT T0120  ; 1#延时使用时间
AND SK2_2  ; 选择行程
OUT YV31  ; 自动化气源1#
LD TR1
AND 66.03  ; 1#延时使用
TIMH(015) 0120 D4081  ; 1#延时使用时间
LD TR0
AND 66.03  ; 1#延时使用
AND 69.03  ; 1#气源用凸轮
DIFU(013) 71.01  ; 1#气源延时起动
; rung 12
LD 64.05  ; 2#使用
OUT TR0
LD 66.05  ; 2#延时使用
AND YV32  ; 自动化气源2#
LD 66.05  ; 2#延时使用
AND 71.02  ; 2#气源延时起动
ORLD
LDNOT 66.05  ; 2#延时使用
AND 69.06  ; 2#气源用凸轮
ORLD
ANDLD
OUT TR1
ANDNOT T0121  ; 2#延时使用时间
AND SK2_2  ; 选择行程
OUT YV32  ; 自动化气源2#
LD TR1
AND 66.05  ; 2#延时使用
TIMH(015) 0121 D4082  ; 2#延时使用时间
LD TR0
AND 66.05  ; 2#延时使用
AND 69.06  ; 2#气源用凸轮
DIFU(013) 71.02  ; 2#气源延时起动

### Section 操作提示

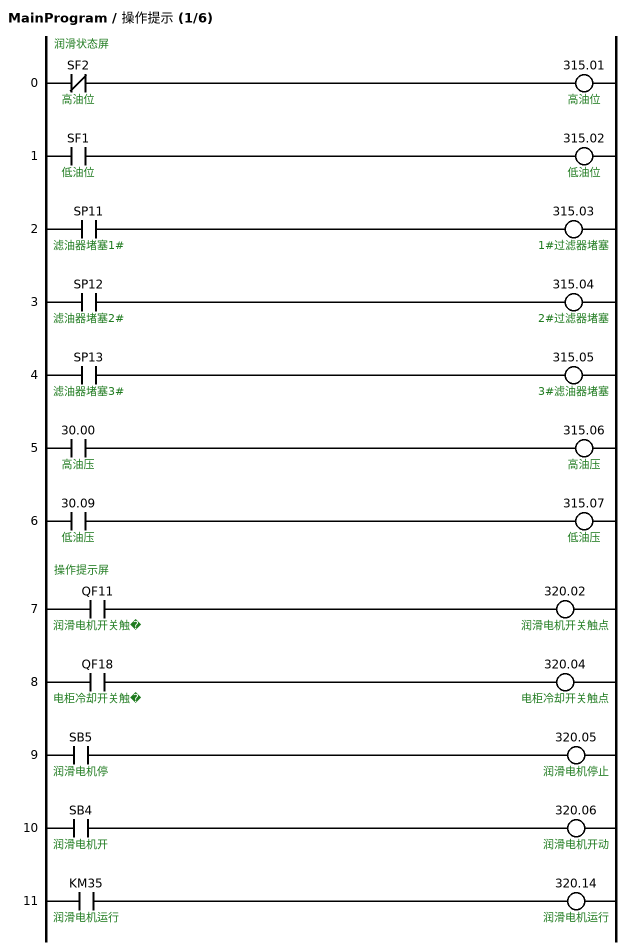
; rung 0: 润滑状态屏
LDNOT SF2  ; 高油位
OUT 315.01  ; 高油位
; rung 1
LD SF1  ; 低油位
OUT 315.02  ; 低油位
; rung 2
LD SP11  ; 滤油器堵塞1#
OUT 315.03  ; 1#过滤器堵塞
; rung 3
LD SP12  ; 滤油器堵塞2#
OUT 315.04  ; 2#过滤器堵塞
; rung 4
LD SP13  ; 滤油器堵塞3#
OUT 315.05  ; 3#滤油器堵塞
; rung 5
LD 30.00  ; 高油压
OUT 315.06  ; 高油压
; rung 6
LD 30.09  ; 低油压
OUT 315.07  ; 低油压
; rung 7: 操作提示屏
LD QF11  ; 润滑电机开关触�
OUT 320.02  ; 润滑电机开关触点
; rung 8
LD QF18  ; 电柜冷却开关触�
OUT 320.04  ; 电柜冷却开关触点
; rung 9
LD SB5  ; 润滑电机停
OUT 320.05  ; 润滑电机停止
; rung 10
LD SB4  ; 润滑电机开
OUT 320.06  ; 润滑电机开动
; rung 11
LD KM35  ; 润滑电机运行
OUT 320.14  ; 润滑电机运行

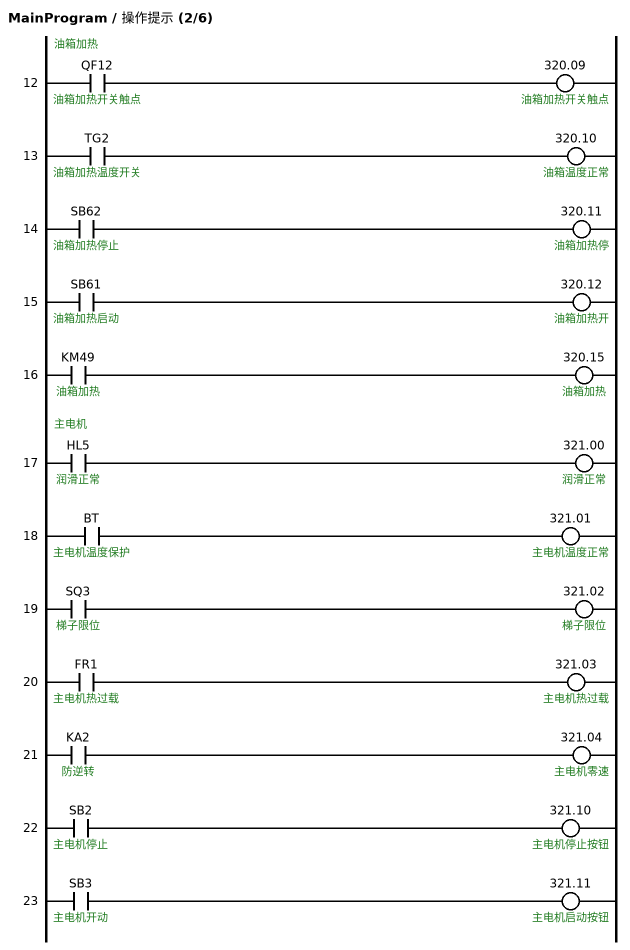
; rung 12: 油箱加热
LD QF12  ; 油箱加热开关触点
OUT 320.09  ; 油箱加热开关触点
; rung 13
LD TG2  ; 油箱加热温度开关
OUT 320.10  ; 油箱温度正常
; rung 14
LD SB62  ; 油箱加热停止
OUT 320.11  ; 油箱加热停
; rung 15
LD SB61  ; 油箱加热启动
OUT 320.12  ; 油箱加热开
; rung 16
LD KM49  ; 油箱加热
OUT 320.15  ; 油箱加热
; rung 17: 主电机
LD HL5  ; 润滑正常
OUT 321.00  ; 润滑正常
; rung 18
LD BT  ; 主电机温度保护
OUT 321.01  ; 主电机温度正常
; rung 19
LD SQ3  ; 梯子限位
OUT 321.02  ; 梯子限位
; rung 20
LD FR1  ; 主电机热过载
OUT 321.03  ; 主电机热过载
; rung 21
LD KA2  ; 防逆转
OUT 321.04  ; 主电机零速
; rung 22
LD SB2  ; 主电机停止
OUT 321.10  ; 主电机停止按钮
; rung 23
LD SB3  ; 主电机开动
OUT 321.11  ; 主电机启动按钮

